DATA_BLOCK "ST10_Flow6_FixtureCodeScan_iDB"
VAR
  sCtrlMode : "SysFlowCtrlGraph";
  sUpdMES_Data : Bool;
  "工件放行中" : Bool;
  "前站站号" : UInt;
  "本站站号" : UInt;
  "弹窗Temp" : Array[1..10] of Int;
  AlarmID : Int;
  TON : Array[0..10] of TON_TIME;
  TOF : Array[0..10] of TOF_TIME;
  sUP : Array[0..10] of Bool;
  "更新RFID完成" : Bool;
  RT_DATA : G7_RTDataPlus_V6;
  Trans1 : G7_TransitionPlus_V6;
  Trans2 : G7_TransitionPlus_V6;
  Trans3 : G7_TransitionPlus_V6;
  Trans325 : G7_TransitionPlus_V6;
  Trans10 : G7_TransitionPlus_V6;
  Trans7 : G7_TransitionPlus_V6;
  Trans102 : G7_TransitionPlus_V6;
  Trans200 : G7_TransitionPlus_V6;
  "Fixture NG" : G7_TransitionPlus_V6;
  R1MaintenReady : G7_TransitionPlus_V6;
  "105ALL Empty" : G7_TransitionPlus_V6;
  TaskMainten : G7_TransitionPlus_V6;
  Trans145 : G7_TransitionPlus_V6;
  R2ScanOk : G7_TransitionPlus_V6;
  Trans147 : G7_TransitionPlus_V6;
  FixtureOk : G7_TransitionPlus_V6;
  Trans250 : G7_TransitionPlus_V6;
  ReadOK_1 : G7_TransitionPlus_V6;
  Trans279 : G7_TransitionPlus_V6;
  Trans282 : G7_TransitionPlus_V6;
  Trans284 : G7_TransitionPlus_V6;
  Trans283 : G7_TransitionPlus_V6;
  ReadOK_8 : G7_TransitionPlus_V6;
  Trans285 : G7_TransitionPlus_V6;
  ReadOK_2 : G7_TransitionPlus_V6;
  ReadOK_7 : G7_TransitionPlus_V6;
  Trans286 : G7_TransitionPlus_V6;
  Trans287 : G7_TransitionPlus_V6;
  Trans288 : G7_TransitionPlus_V6;
  Trans291 : G7_TransitionPlus_V6;
  ReadOK_3 : G7_TransitionPlus_V6;
  Trans289 : G7_TransitionPlus_V6;
  Trans292 : G7_TransitionPlus_V6;
  Trans293 : G7_TransitionPlus_V6;
  Trans280 : G7_TransitionPlus_V6;
  Trans295 : G7_TransitionPlus_V6;
  ReadOK_4 : G7_TransitionPlus_V6;
  Trans302 : G7_TransitionPlus_V6;
  Trans290 : G7_TransitionPlus_V6;
  ReadOK_9 : G7_TransitionPlus_V6;
  Trans294 : G7_TransitionPlus_V6;
  Trans310 : G7_TransitionPlus_V6;
  Trans311 : G7_TransitionPlus_V6;
  Trans296 : G7_TransitionPlus_V6;
  Trans297 : G7_TransitionPlus_V6;
  Trans298 : G7_TransitionPlus_V6;
  Trans309 : G7_TransitionPlus_V6;
  Trans312 : G7_TransitionPlus_V6;
  ReadOK_19 : G7_TransitionPlus_V6;
  Trans336 : G7_TransitionPlus_V6;
  Trans299 : G7_TransitionPlus_V6;
  Trans307 : G7_TransitionPlus_V6;
  ReadOK_5 : G7_TransitionPlus_V6;
  ReadOK_18 : G7_TransitionPlus_V6;
  "317GripScanng" : G7_TransitionPlus_V6;
  Trans349 : G7_TransitionPlus_V6;
  "319GripScanOK" : G7_TransitionPlus_V6;
  ReadOK_24 : G7_TransitionPlus_V6;
  Trans300 : G7_TransitionPlus_V6;
  Trans301 : G7_TransitionPlus_V6;
  Trans303 : G7_TransitionPlus_V6;
  Trans304 : G7_TransitionPlus_V6;
  ReadOK_6 : G7_TransitionPlus_V6;
  Trans308 : G7_TransitionPlus_V6;
  Trans348 : G7_TransitionPlus_V6;
  Trans305 : G7_TransitionPlus_V6;
  Trans350 : G7_TransitionPlus_V6;
  Trans306 : G7_TransitionPlus_V6;
  ReadOK_10 : G7_TransitionPlus_V6;
  Trans352 : G7_TransitionPlus_V6;
  Trans353 : G7_TransitionPlus_V6;
  ReadOK_14 : G7_TransitionPlus_V6;
  Trans313 : G7_TransitionPlus_V6;
  Trans315 : G7_TransitionPlus_V6;
  R3ScanOk : G7_TransitionPlus_V6;
  Trans314 : G7_TransitionPlus_V6;
  Trans316 : G7_TransitionPlus_V6;
  ReadOK_11 : G7_TransitionPlus_V6;
  Trans317 : G7_TransitionPlus_V6;
  Trans321 : G7_TransitionPlus_V6;
  Trans318 : G7_TransitionPlus_V6;
  ReadOK_15 : G7_TransitionPlus_V6;
  Trans326 : G7_TransitionPlus_V6;
  Trans319 : G7_TransitionPlus_V6;
  Trans320 : G7_TransitionPlus_V6;
  ReadOK_12 : G7_TransitionPlus_V6;
  Trans329 : G7_TransitionPlus_V6;
  Trans330 : G7_TransitionPlus_V6;
  Trans322 : G7_TransitionPlus_V6;
  "Robot1AllScan NG" : G7_TransitionPlus_V6;
  ReadOK_16 : G7_TransitionPlus_V6;
  Trans323 : G7_TransitionPlus_V6;
  Trans324 : G7_TransitionPlus_V6;
  ReadOK_13 : G7_TransitionPlus_V6;
  Trans331 : G7_TransitionPlus_V6;
  Trans332 : G7_TransitionPlus_V6;
  Trans327 : G7_TransitionPlus_V6;
  Trans333 : G7_TransitionPlus_V6;
  ReadOK_17 : G7_TransitionPlus_V6;
  Trans328 : G7_TransitionPlus_V6;
  Trans334 : G7_TransitionPlus_V6;
  Trans335 : G7_TransitionPlus_V6;
  ReadOK_20 : G7_TransitionPlus_V6;
  Trans337 : G7_TransitionPlus_V6;
  Trans338 : G7_TransitionPlus_V6;
  Trans339 : G7_TransitionPlus_V6;
  ReadOK_21 : G7_TransitionPlus_V6;
  Trans340 : G7_TransitionPlus_V6;
  Trans341 : G7_TransitionPlus_V6;
  Trans342 : G7_TransitionPlus_V6;
  ReadOK_22 : G7_TransitionPlus_V6;
  Trans343 : G7_TransitionPlus_V6;
  Trans344 : G7_TransitionPlus_V6;
  Trans345 : G7_TransitionPlus_V6;
  ReadOK_23 : G7_TransitionPlus_V6;
  Trans346 : G7_TransitionPlus_V6;
  Trans400 : G7_TransitionPlus_V6;
  Trans347 : G7_TransitionPlus_V6;
  Trans371 : G7_TransitionPlus_V6;
  Trans403 : G7_TransitionPlus_V6;
  R3ScanNG : G7_TransitionPlus_V6;
  Trans405 : G7_TransitionPlus_V6;
  GripScanNG1 : G7_TransitionPlus_V6;
  GripScanOK : G7_TransitionPlus_V6;
  Trans413 : G7_TransitionPlus_V6;
  Trans414 : G7_TransitionPlus_V6;
  ChengeOk : G7_TransitionPlus_V6;
  Trans416 : G7_TransitionPlus_V6;
  TypeChange : G7_TransitionPlus_V6;
  Trans418 : G7_TransitionPlus_V6;
  Trans419 : G7_TransitionPlus_V6;
  Trans420 : G7_TransitionPlus_V6;
  Trans421 : G7_TransitionPlus_V6;
  Trans422 : G7_TransitionPlus_V6;
  Trans423 : G7_TransitionPlus_V6;
  Trans606 : G7_TransitionPlus_V6;
  Trans613 : G7_TransitionPlus_V6;
  Trans608 : G7_TransitionPlus_V6;
  "Robot1AllScan Ok" : G7_TransitionPlus_V6;
  Trans612 : G7_TransitionPlus_V6;
  Trans614 : G7_TransitionPlus_V6;
  Trans615 : G7_TransitionPlus_V6;
  Trans616 : G7_TransitionPlus_V6;
  Trans617 : G7_TransitionPlus_V6;
  Trans620 : G7_TransitionPlus_V6;
  Trans684 : G7_TransitionPlus_V6;
  Trans607 : G7_TransitionPlus_V6;
  Trans629 : G7_TransitionPlus_V6;
  Trans630 : G7_TransitionPlus_V6;
  Trans631 : G7_TransitionPlus_V6;
  Trans632 : G7_TransitionPlus_V6;
  Trans633 : G7_TransitionPlus_V6;
  Trans634 : G7_TransitionPlus_V6;
  Trans635 : G7_TransitionPlus_V6;
  Trans636 : G7_TransitionPlus_V6;
  Trans637 : G7_TransitionPlus_V6;
  Trans638 : G7_TransitionPlus_V6;
  Trans642 : G7_TransitionPlus_V6;
  Trans652 : G7_TransitionPlus_V6;
  Trans653 : G7_TransitionPlus_V6;
  Trans673 : G7_TransitionPlus_V6;
  Trans675 : G7_TransitionPlus_V6;
  Trans609 : G7_TransitionPlus_V6;
  Trans676 : G7_TransitionPlus_V6;
  Trans618 : G7_TransitionPlus_V6;
  Trans619 : G7_TransitionPlus_V6;
  Trans677 : G7_TransitionPlus_V6;
  Trans621 : G7_TransitionPlus_V6;
  Trans622 : G7_TransitionPlus_V6;
  Trans623 : G7_TransitionPlus_V6;
  Trans610 : G7_TransitionPlus_V6;
  Trans639 : G7_TransitionPlus_V6;
  Trans640 : G7_TransitionPlus_V6;
  Trans641 : G7_TransitionPlus_V6;
  Trans643 : G7_TransitionPlus_V6;
  Trans644 : G7_TransitionPlus_V6;
  Trans645 : G7_TransitionPlus_V6;
  Trans646 : G7_TransitionPlus_V6;
  Trans647 : G7_TransitionPlus_V6;
  Trans648 : G7_TransitionPlus_V6;
  Trans649 : G7_TransitionPlus_V6;
  Trans624 : G7_TransitionPlus_V6;
  Trans685 : G7_TransitionPlus_V6;
  Trans674 : G7_TransitionPlus_V6;
  R2ScanNG : G7_TransitionPlus_V6;
  Trans678 : G7_TransitionPlus_V6;
  Trans625 : G7_TransitionPlus_V6;
  Trans626 : G7_TransitionPlus_V6;
  Trans627 : G7_TransitionPlus_V6;
  Trans650 : G7_TransitionPlus_V6;
  Trans655 : G7_TransitionPlus_V6;
  Trans656 : G7_TransitionPlus_V6;
  Trans657 : G7_TransitionPlus_V6;
  Trans659 : G7_TransitionPlus_V6;
  ALLScanOk : G7_TransitionPlus_V6;
  Trans661 : G7_TransitionPlus_V6;
  Trans662 : G7_TransitionPlus_V6;
  Trans663 : G7_TransitionPlus_V6;
  Trans664 : G7_TransitionPlus_V6;
  FixtureAllOk : G7_TransitionPlus_V6;
  Trans720 : G7_TransitionPlus_V6;
  Trans740 : G7_TransitionPlus_V6;
  FixtureNG : G7_TransitionPlus_V6;
  F6_Initial : G7_StepPlus_V6;
  S2 : G7_StepPlus_V6;
  S3 : G7_StepPlus_V6;
  S4 : G7_StepPlus_V6;
  S5_MESInitial : G7_StepPlus_V6;
  S8 : G7_StepPlus_V6;
  S9 : G7_StepPlus_V6;
  S10_InitialFinish : G7_StepPlus_V6;
  ProcessStart : G7_StepPlus_V6;
  "Determine TableFixtureStatus" : G7_StepPlus_V6;
  RobotMaintenanceReq : G7_StepPlus_V6;
  WaitAllPartEmpty : G7_StepPlus_V6;
  ToolScanCondition : G7_StepPlus_V6;
  Robot2CheckScanResult : G7_StepPlus_V6;
  "Fixturecode reading" : G7_StepPlus_V6;
  CheckScanStatus : G7_StepPlus_V6;
  "RB1_Process scan" : G7_StepPlus_V6;
  DataMove_1 : G7_StepPlus_V6;
  DataMove_2 : G7_StepPlus_V6;
  "Start 1st reading" : G7_StepPlus_V6;
  "Check reader Ready" : G7_StepPlus_V6;
  "Wait reading complete" : G7_StepPlus_V6;
  "Start 2st reading" : G7_StepPlus_V6;
  "Check reader Ready_1" : G7_StepPlus_V6;
  "Wait reading complete_1" : G7_StepPlus_V6;
  DataMove_3 : G7_StepPlus_V6;
  "Start 3st reading" : G7_StepPlus_V6;
  "Check reader Ready_2" : G7_StepPlus_V6;
  "Wait reading complete_2" : G7_StepPlus_V6;
  DataMove_4 : G7_StepPlus_V6;
  "Start 4st reading" : G7_StepPlus_V6;
  "Check reader Ready_3" : G7_StepPlus_V6;
  "Wait reading complete_3" : G7_StepPlus_V6;
  DataMove_7 : G7_StepPlus_V6;
  DataMove_5 : G7_StepPlus_V6;
  "Start 5st reading" : G7_StepPlus_V6;
  "Check reader Ready_4" : G7_StepPlus_V6;
  "Wait reading complete_4" : G7_StepPlus_V6;
  DataMove_8 : G7_StepPlus_V6;
  DataMove_6 : G7_StepPlus_V6;
  "Start 6st reading" : G7_StepPlus_V6;
  "Check reader Ready_5" : G7_StepPlus_V6;
  "Wait reading complete_5" : G7_StepPlus_V6;
  "Start 1st reading_1" : G7_StepPlus_V6;
  "Check reader Ready_6" : G7_StepPlus_V6;
  "Wait reading complete_6" : G7_StepPlus_V6;
  "Start 5st reading_1" : G7_StepPlus_V6;
  "Check reader Ready_7" : G7_StepPlus_V6;
  "Wait reading complete_7" : G7_StepPlus_V6;
  "Wait reading complete_10" : G7_StepPlus_V6;
  DataMove_10 : G7_StepPlus_V6;
  "Wait reading complete_14" : G7_StepPlus_V6;
  "Start 5st reading_2" : G7_StepPlus_V6;
  RobotScanGripPos1Comp : G7_StepPlus_V6;
  Robot2FixtrueScanStart : G7_StepPlus_V6;
  "Wait reading complete_8" : G7_StepPlus_V6;
  "Check reader Ready_8" : G7_StepPlus_V6;
  DataMove_14 : G7_StepPlus_V6;
  WaitRobotScanGripPos2Reach : G7_StepPlus_V6;
  RobotScanGripPos1Comp_1 : G7_StepPlus_V6;
  Robot2StartScan : G7_StepPlus_V6;
  WaitRobotScanGripPos2Reach_1 : G7_StepPlus_V6;
  Robot1ToMaintenance : G7_StepPlus_V6;
  DataMove_9 : G7_StepPlus_V6;
  DataMove_18 : G7_StepPlus_V6;
  WaitRobotScanStart : G7_StepPlus_V6;
  RequestRobotScanFixture : G7_StepPlus_V6;
  "Start 4st reading_1" : G7_StepPlus_V6;
  "Check reader Ready_9" : G7_StepPlus_V6;
  "Wait reading complete_9" : G7_StepPlus_V6;
  WaitRobotScanPos1Reach : G7_StepPlus_V6;
  CheckRobot1ScanResult : G7_StepPlus_V6;
  "Check reader Ready_18" : G7_StepPlus_V6;
  "Wait reading complete_18" : G7_StepPlus_V6;
  DataMove_19 : G7_StepPlus_V6;
  "Start 3st reading_1" : G7_StepPlus_V6;
  "Start 2st reading_1" : G7_StepPlus_V6;
  Robot3CheckScanResult : G7_StepPlus_V6;
  WaitRobotScanPos1Reach_3 : G7_StepPlus_V6;
  "Wait reading complete_19" : G7_StepPlus_V6;
  DataMove_20 : G7_StepPlus_V6;
  RobotScanGripPos1Comp_2 : G7_StepPlus_V6;
  WaitRobotScanGripPos2Reach_2 : G7_StepPlus_V6;
  WaitRobotScanGripPos1Reach : G7_StepPlus_V6;
  WaitRobotScanPos2Reach : G7_StepPlus_V6;
  "Check reader Ready_10" : G7_StepPlus_V6;
  WaitRobotScanPos3Reach : G7_StepPlus_V6;
  "Start 10st reading" : G7_StepPlus_V6;
  WaitRobotScanPos4Reach : G7_StepPlus_V6;
  Robot1FixtureScan : G7_StepPlus_V6;
  WaitRobotScanPos5Reach : G7_StepPlus_V6;
  "Check reader Ready_11" : G7_StepPlus_V6;
  WaitRobotScanPos1Reach_1 : G7_StepPlus_V6;
  "Start 11st reading" : G7_StepPlus_V6;
  WaitRobotScanPos7Reach : G7_StepPlus_V6;
  "Check reader Ready_14" : G7_StepPlus_V6;
  "Wait reading complete_11" : G7_StepPlus_V6;
  DataMove_11 : G7_StepPlus_V6;
  "Start 10st reading_1" : G7_StepPlus_V6;
  RobotScanGripPos2Comp : G7_StepPlus_V6;
  WaitRobotScanGripPos3Reach : G7_StepPlus_V6;
  "Check reader Ready_12" : G7_StepPlus_V6;
  "Start 11st reading_1" : G7_StepPlus_V6;
  "Check reader Ready_23" : G7_StepPlus_V6;
  "Wait reading complete_12" : G7_StepPlus_V6;
  DataMove_12 : G7_StepPlus_V6;
  "Check reader Ready_15" : G7_StepPlus_V6;
  RobotScanGripPos3Comp : G7_StepPlus_V6;
  WaitRobotScanGripPos4Reach : G7_StepPlus_V6;
  "Check reader Ready_13" : G7_StepPlus_V6;
  "Start 11st reading_2" : G7_StepPlus_V6;
  "Start 11st reading_3" : G7_StepPlus_V6;
  "Wait reading complete_13" : G7_StepPlus_V6;
  DataMove_13 : G7_StepPlus_V6;
  "Wait reading complete_15" : G7_StepPlus_V6;
  RobotScanGripPos4Comp : G7_StepPlus_V6;
  DataMove_15 : G7_StepPlus_V6;
  StartRobotScanGripperCode : G7_StepPlus_V6;
  RobotScanGripperReachPos1 : G7_StepPlus_V6;
  Robot3StartToScan : G7_StepPlus_V6;
  Robot2StartToMaintenanc : G7_StepPlus_V6;
  WaitRobotScanPos1Reach_2 : G7_StepPlus_V6;
  WaitRobotScanPos5Reach_1 : G7_StepPlus_V6;
  WaitRobotScanPos2Reach_1 : G7_StepPlus_V6;
  WaitRobotScanPos4Reach_1 : G7_StepPlus_V6;
  RobotScanGripPos2Comp_1 : G7_StepPlus_V6;
  WaitRobotScanGripPos3Reach_1 : G7_StepPlus_V6;
  "Check reader Ready_16" : G7_StepPlus_V6;
  "Start 11st reading_4" : G7_StepPlus_V6;
  "Wait reading complete_16" : G7_StepPlus_V6;
  DataMove_16 : G7_StepPlus_V6;
  WaitRobotScanPos3Reach_1 : G7_StepPlus_V6;
  RobotScanGripPos3Comp_1 : G7_StepPlus_V6;
  RequestRobotScan_1 : G7_StepPlus_V6;
  WaitRobotScanGripPos1Reach_1 : G7_StepPlus_V6;
  "Check reader Ready_19" : G7_StepPlus_V6;
  "Start 10st reading_2" : G7_StepPlus_V6;
  WaitRobotScanGripPos4Reach_1 : G7_StepPlus_V6;
  "Check reader Ready_20" : G7_StepPlus_V6;
  "Check reader Ready_17" : G7_StepPlus_V6;
  "Start 11st reading_5" : G7_StepPlus_V6;
  "Start 11st reading_6" : G7_StepPlus_V6;
  "Wait reading complete_17" : G7_StepPlus_V6;
  DataMove_17 : G7_StepPlus_V6;
  "Wait reading complete_20" : G7_StepPlus_V6;
  RobotScanGripPos4Comp_1 : G7_StepPlus_V6;
  DataMove_21 : G7_StepPlus_V6;
  RobotScanGripPos2Comp_2 : G7_StepPlus_V6;
  WaitRobotScanGripPos3Reach_2 : G7_StepPlus_V6;
  "Check reader Ready_21" : G7_StepPlus_V6;
  "Start 11st reading_7" : G7_StepPlus_V6;
  "Wait reading complete_21" : G7_StepPlus_V6;
  DataMove_22 : G7_StepPlus_V6;
  RobotScanGripPos3Comp_2 : G7_StepPlus_V6;
  Robot3FixtrueScanStart : G7_StepPlus_V6;
  WaitRobotScanGripPos4Reach_2 : G7_StepPlus_V6;
  "Check reader Ready_22" : G7_StepPlus_V6;
  "Start 11st reading_8" : G7_StepPlus_V6;
  "Wait reading complete_22" : G7_StepPlus_V6;
  DataMove_23 : G7_StepPlus_V6;
  RobotScanGripPos4Comp_2 : G7_StepPlus_V6;
  WaitRobot2ScanFinishAndInHome : G7_StepPlus_V6;
  AllScanFinish : G7_StepPlus_V6;
  Robot3StartToMaintenance : G7_StepPlus_V6;
  Robot2CheckScanStatus : G7_StepPlus_V6;
  Robot3CheckScanStatus : G7_StepPlus_V6;
  WaitRobotScanPos1Reach_4 : G7_StepPlus_V6;
  "Wait reading complete_23" : G7_StepPlus_V6;
  DataMove_24 : G7_StepPlus_V6;
  CheckStationEmpty : G7_StepPlus_V6;
  ClearAllBeltPallet : G7_StepPlus_V6;
  CheckTypeChenge : G7_StepPlus_V6;
  TypeCheckOk : G7_StepPlus_V6;
  CheckTypeTrigger : G7_StepPlus_V6;
  ResetChangeOverReq : G7_StepPlus_V6;
  WaitServoStop : G7_StepPlus_V6;
  "WaitRobotBRAKETEST and MASTERINGTEST finish" : G7_StepPlus_V6;
  MaintenanceProcess : G7_StepPlus_V6;
  ReqRobotToMantenPos : G7_StepPlus_V6;
  WaitR1MaintenPosFinsh : G7_StepPlus_V6;
  Robot2ToMaintenance : G7_StepPlus_V6;
  MaintenanceProcess_1 : G7_StepPlus_V6;
  ReqRobotToMantenPos_1 : G7_StepPlus_V6;
  WaitR1MaintenPosFinsh_1 : G7_StepPlus_V6;
  Robot3ToMaintenance : G7_StepPlus_V6;
  MaintenanceProcess_2 : G7_StepPlus_V6;
  ReqRobotToMantenPos_2 : G7_StepPlus_V6;
  WaitR1MaintenPosFinsh_2 : G7_StepPlus_V6;
  CycleEnd_2 : G7_StepPlus_V6;
  Step720 : G7_StepPlus_V6;
  Step712 : G7_StepPlus_V6;
END_VAR
BEGIN
END_DATA_BLOCK
